(* CODESYS project SPT_NC_Homing.library
   Company: Beckhoff Automation LLC
   DefaultNamespace: SPT_NCHoming
   Version: 3.0.1
   Placeholder: SPT NC Homing
   Title: SPT NC Homing

Project tree, tasks and I/O mapping:
  libraries: SPT Base Types, * (Beckhoff Automation LLC); SPT NC Axis, * (Beckhoff Automation LLC); Tc2_MC2, * (Beckhoff Automation GmbH); Tc2_Standard, * (Beckhoff Automation GmbH); Tc3_MC2_AdvancedHoming, * (Beckhoff Automation GmbH); Tc3_Module, * (Beckhoff Automation GmbH); Tc3_System, * (Beckhoff Automation GmbH)
  DUTs/
    data type ST_AbsHomeParameters
    data type ST_StepBlockLagBasedParameters
  Function Blocks/
    function block FB_HomeRoutine_AbsHoming [ST]: Axis, CyclicLogic, Execute, Parameters
    function block FB_HomeRoutine_HardStop [ST]: Axis, CyclicLogic, Execute, HomePosition, Parameters
    function block FB_HomeRoutine_SetPosition [ST]: Axis, CyclicLogic, Execute, HomePosition
    function block FB_HomeRoutine_SetZeroHere [ST]: Axis, CyclicLogic, Execute
  Project Information/
    function F_GetCompany [ST]
    function F_GetTitle [ST]
    function F_GetVersion [ST]
  Version/
    global variables Global_Version
*)

// DUTs/ST_AbsHomeParameters
TYPE ST_AbsHomeParameters :
    STRUCT
        PositionBias           : LREAL;
        PositionLimit_Positive : LREAL;
        PositionLimit_Negative : LREAL;
    END_STRUCT
END_TYPE

// DUTs/ST_StepBlockLagBasedParameters
TYPE ST_StepBlockLagBasedParameters :
    STRUCT
        Direction              : MC_Home_Direction := mcNegativeDirection;
        Velocity               : LREAL             := 10;
        Acceleration           : LREAL             := 100;
        Deceleration           : LREAL             := 100;
        Jerk                   : LREAL             := 1000;
        DetectionVelocityLimit : LREAL             := 5;
        DetectionVelocityTime  : TIME              := T#500MS;
        TimeLimit              : TIME;
        DistanceLimit          : LREAL;
        TorqueLimit            : LREAL            := 10;
        LagLimit               : LREAL            := 10;
        Options                : ST_Home_Options3 := (InstantLagReduction := TRUE);
    END_STRUCT
END_TYPE

// Version/Global_Version
{attribute 'TcGenerated'}
{attribute 'no-analysis'}
{attribute 'linkalways'}
// This function has been automatically generated from the project information.
VAR_GLOBAL CONSTANT
	{attribute 'const_non_replaced'}
	stLibVersion_SPT_NC_Homing : ST_LibVersion := (iMajor := 3, iMinor := 0, iBuild := 1, iRevision := 0, nFlags := 1, sVersion := '3.0.1');
END_VAR

// Function Blocks/FB_HomeRoutine_AbsHoming
FUNCTION_BLOCK FB_HomeRoutine_AbsHoming EXTENDS FB_CyclicFB IMPLEMENTS I_MotionSequence
VAR
    _Axis : I_BasicAxis;
END_VAR

VAR
    _HomingDn                 : BOOL;
    _Reset                    : BOOL;
    _Parameters               : REFERENCE TO ST_AbsHomeParameters;
    SequenceStep              : UDINT;
    ReadWatchdog              : TON;
    WriteWatchdog             : TON;
    McReadParameter_Bias      : MC_ReadParameter;
    McWriteParameter_Bias     : MC_WriteParameter;
    McWriteParameter_SwPosLim : MC_WriteParameter;
    McWriteParameter_SwNegLim : MC_WriteParameter;
    McHome                    : MC_Home;
    CurrentPositionBias       : LREAL;
END_VAR

//There should be no code in the function block body

PROPERTY Axis : I_BasicAxis
GET
Axis := _Axis;
END_GET
SET
_Axis := Axis;
END_SET
END_PROPERTY

METHOD CyclicLogic
VAR_INPUT
END_VAR
IF __ISVALIDREF(_Parameters) THEN
    CASE SequenceStep OF
        0: (* Init State *)
            _Busy                             := TRUE;
            ReadWatchdog.IN                   := FALSE;
            WriteWatchdog.IN                  := TRUE;
            McReadParameter_Bias.Enable       := FALSE;
            McWriteParameter_Bias.Execute     := TRUE;
            McWriteParameter_SwPosLim.Execute := TRUE;
            McWriteParameter_SwNegLim.Execute := TRUE;
            SequenceStep                      := 10;
        10: (* Wait for init done *)

            // check for errors
            IF WriteWatchdog.Q THEN
                SequenceStep := 500;
                _Error       := TRUE;
                _ErrorID     := 10;
            ELSIF McWriteParameter_Bias.Error THEN
                SequenceStep := 500;
                _Error       := TRUE;
                _ErrorID     := McWriteParameter_Bias.ErrorID;
            ELSIF McWriteParameter_SwPosLim.Error THEN
                SequenceStep := 500;
                _Error       := TRUE;
                _ErrorID     := McWriteParameter_SwPosLim.ErrorID;
            ELSIF McWriteParameter_SwNegLim.Error THEN
                SequenceStep := 500;
                _Error       := TRUE;
                _ErrorID     := McWriteParameter_SwNegLim.ErrorID;
            END_IF

            IF (McWriteParameter_Bias.Done AND McWriteParameter_SwPosLim.Done AND McWriteParameter_SwNegLim.Done) THEN
                WriteWatchdog.IN := FALSE;
                McHome.Execute   := TRUE;
                _Busy            := FALSE;
            END_IF
        20: (* Reads the Position Bias Variable *)
            _Busy                             := TRUE;
            WriteWatchdog.IN                  := FALSE;
            McWriteParameter_Bias.Execute     := FALSE;
            McWriteParameter_SwPosLim.Execute := FALSE;
            McWriteParameter_SwNegLim.Execute := FALSE;

            (* 1042 = Axis Encoder Offset ... AKA: Position Bias *)
            IF NOT McReadParameter_Bias.Enable THEN
                ReadWatchdog.IN             := TRUE;
                McReadParameter_Bias.Enable := TRUE;
            END_IF

            IF (McReadParameter_Bias.Enable AND McReadParameter_Bias.Valid) THEN
                ReadWatchdog.IN             := FALSE;
                McReadParameter_Bias.Enable := FALSE;

                (* Do the calculations to figure how far to adjust the Position Bias # *)

                (* Write Value back to the bias for the new teach position *)
                _Parameters.PositionBias := CurrentPositionBias + (_Axis.Axis.NcToPlc.ActPos * -1.0);
                SequenceStep             := 30;
            ELSIF McReadParameter_Bias.Error THEN
                SequenceStep := 500;
                _Error       := TRUE;
                _ErrorID     := McReadParameter_Bias.ErrorID;
            ELSIF ReadWatchdog.Q THEN
                SequenceStep := 500;
                _Error       := TRUE;
                _ErrorID     := 20;
            END_IF
        30:
            _Busy                             := TRUE;
            WriteWatchdog.IN                  := TRUE;
            McWriteParameter_Bias.Execute     := TRUE;
            McWriteParameter_SwPosLim.Execute := TRUE;
            McWriteParameter_SwNegLim.Execute := TRUE;
            SequenceStep                      := 10;
        500: (* Error State *)
            _Busy                             := FALSE;
            ReadWatchdog.IN                   := FALSE;
            WriteWatchdog.IN                  := FALSE;
            McReadParameter_Bias.Enable       := FALSE;
            McWriteParameter_Bias.Execute     := FALSE;
            McWriteParameter_SwPosLim.Execute := FALSE;
            McWriteParameter_SwNegLim.Execute := FALSE;
    END_CASE
ELSE
    _Busy                             := FALSE;
    _Error                            := FALSE;
    _ErrorID                          := 0;
    SequenceStep                      := 0;
    ReadWatchdog.IN                   := FALSE;
    WriteWatchdog.IN                  := FALSE;
    McReadParameter_Bias.Enable       := FALSE;
    McWriteParameter_Bias.Execute     := FALSE;
    McWriteParameter_SwPosLim.Execute := FALSE;
    McWriteParameter_SwNegLim.Execute := FALSE;
END_IF

ReadWatchdog(PT := T#1S);
WriteWatchdog(PT := T#1S);
McHome(Axis := _Axis.Axis, HomingMode := MC_ForceCalibration);

(* Position Bias Reading *)
McReadParameter_Bias(ParameterNumber := MC_AxisParameter.AxisEncoderOffset, (*AxisEncoderOffset*)
                     Axis            := _Axis.Axis,
                     Value           => CurrentPositionBias);

(* Writes the Position Bias Variable *)
McWriteParameter_Bias(Execute         := McWriteParameter_Bias.Execute,
                      ParameterNumber := MC_AxisParameter.AxisEncoderOffset, (*AxisEncoderOffset*)
                      Value           := _Parameters.PositionBias,
                      Axis            := _Axis.Axis);

(* Writes the SW Positive Limit Variable *)
McWriteParameter_SwPosLim(Execute         := McWriteParameter_SwPosLim.Execute,
                          ParameterNumber := MC_AxisParameter.SWLimitPos,
                          Value           := _Parameters.PositionLimit_Positive,
                          Axis            := _Axis.Axis);

(* Writes the SW Negetive Limit Variable *)
McWriteParameter_SwNegLim(Execute         := McWriteParameter_SwNegLim.Execute,
                          ParameterNumber := MC_AxisParameter.SWLimitNeg,
                          Value           := _Parameters.PositionLimit_Negative,
                          Axis            := _Axis.Axis);
END_METHOD

METHOD Execute : BOOL
IF (_Axis = 0) OR _Busy OR NOT (McWriteParameter_Bias.Done AND McWriteParameter_SwPosLim.Done AND McWriteParameter_SwNegLim.Done) THEN
    RETURN;
END_IF

_Busy        := TRUE;
_Error       := FALSE;
_ErrorID     := 0;
_HomingDn    := FALSE;
SequenceStep := 20;
Execute      := TRUE;
END_METHOD

PROPERTY Parameters : REFERENCE TO ST_AbsHomeParameters
GET
IF __ISVALIDREF(_Parameters) THEN
    Parameters REF= _Parameters;
END_IF
END_GET
SET
_Parameters ref= Parameters;
END_SET
END_PROPERTY

END_FUNCTION_BLOCK

// Function Blocks/FB_HomeRoutine_HardStop
FUNCTION_BLOCK FINAL FB_HomeRoutine_HardStop EXTENDS FB_CyclicFB IMPLEMENTS I_MotionSequence
VAR
    _Axis : I_BasicAxis;
END_VAR

VAR
    MCStepBlock    : MC_StepBlockLagBasedDetection;
    MCHomeDirect   : MC_HomeDirect;
    MCReset        : MC_Reset;
    MCAbortHoming  : MC_AbortHoming;
    AxisParameters : MC_HomingParameter;
    _Parameters    : ST_StepBlockLagBasedParameters;
    _HomePosition  : LREAL;
    SequenceStep   : UDINT;
END_VAR

//There should be no code in the function block body

PROPERTY Axis : I_BasicAxis
GET
Axis := _Axis;
END_GET
SET
_Axis := Axis;
END_SET
END_PROPERTY

METHOD PUBLIC CyclicLogic
CASE SequenceStep OF
    10:
        MCStepBlock(Axis                   := _Axis.Axis,
                    Parameter              := AxisParameters,
                    Execute                := TRUE,
                    Direction              := _Parameters.Direction,
                    Velocity               := _Parameters.Velocity,
                    Acceleration           := _Parameters.Acceleration,
                    Deceleration           := _Parameters.Deceleration,
                    Jerk                   := _Parameters.Jerk,
                    DetectionVelocityLimit := _Parameters.DetectionVelocityLimit,
                    DetectionVelocityTime  := _Parameters.DetectionVelocityTime,
                    TimeLimit              := _Parameters.TimeLimit,
                    DistanceLimit          := _Parameters.DistanceLimit,
                    TorqueLimit            := _Parameters.TorqueLimit,
                    LagLimit               := _Parameters.LagLimit,
                    Options                := _Parameters.Options);

        IF NOT MCStepBlock.Busy THEN
            IF MCStepBlock.Error THEN
                _Error       := TRUE;
                _ErrorID     := MCStepBlock.ErrorID;
                SequenceStep := 999;
            ELSE
                //No error occurred
                SequenceStep := SequenceStep + 10;
            END_IF

            MCStepBlock(Axis := _Axis.Axis, Parameter := AxisParameters, Execute := FALSE);
        END_IF
    20:
        MCHomeDirect(Axis        := _Axis.Axis,
                     Parameter   := AxisParameters,
                     Execute     := TRUE,
                     SetPosition := _HomePosition);

        IF NOT MCHomeDirect.Busy THEN
            IF MCHomeDirect.Error THEN
                _Error       := TRUE;
                _ErrorID     := MCHomeDirect.ErrorID;
                SequenceStep := 999;
            END_IF

            //Done
            SequenceStep := 0;
            MCHomeDirect(Axis := _Axis.Axis, Parameter := AxisParameters, Execute := FALSE);
        END_IF
    999:
        //An error occurred above--clear out position lag so we don't fault the axis with AbortHoming
        MCReset(Axis := _Axis.Axis, Execute := TRUE);
        IF NOT MCReset.Busy THEN
            //If this errors there's not much we can do about it
            SequenceStep := 1000;
            MCReset(Axis := _Axis.Axis, Execute := FALSE);
        END_IF
    1000:
        MCAbortHoming(Axis := _Axis.Axis, Parameter := AxisParameters, Execute := TRUE);
        IF NOT MCAbortHoming.Busy THEN
            IF MCAbortHoming.Error THEN
                _Error       := TRUE;
                _ErrorID     := MCAbortHoming.ErrorID;
                SequenceStep := 0;
            ELSE
                //No error occurred
                SequenceStep := 0;
            END_IF

            MCAbortHoming(Axis := _Axis.Axis, Parameter := AxisParameters, Execute := FALSE);
        END_IF
END_CASE

_Busy := SequenceStep <> 0;
END_METHOD

METHOD PUBLIC Execute : BOOL
IF (_Axis = 0) OR _Busy THEN
    RETURN;
END_IF

_Busy        := TRUE;
_Error       := FALSE;
_ErrorID     := 0;
SequenceStep := 10;
Execute      := TRUE;
END_METHOD

PROPERTY HomePosition : LREAL
GET
HomePosition := _HomePosition;
END_GET
SET
_HomePosition := HomePosition;
END_SET
END_PROPERTY

PROPERTY Parameters : ST_StepBlockLagBasedParameters
GET
Parameters := _Parameters;
END_GET
SET
_Parameters := Parameters;
END_SET
END_PROPERTY

END_FUNCTION_BLOCK

// Function Blocks/FB_HomeRoutine_SetPosition
FUNCTION_BLOCK FINAL FB_HomeRoutine_SetPosition EXTENDS FB_CyclicFB IMPLEMENTS I_MotionSequence
VAR_INPUT
END_VAR

VAR_OUTPUT
END_VAR

VAR
    _Axis : I_BasicAxis;
END_VAR

VAR
    MCSetPosition : MC_SetPosition;
END_VAR

//There should be no code in the function block body

PROPERTY Axis : I_BasicAxis
GET
Axis := _Axis;
END_GET
SET
_Axis := Axis;
END_SET
END_PROPERTY

METHOD PUBLIC CyclicLogic
MCSetPosition(Axis := _Axis.Axis, Busy => _Busy);
IF NOT MCSetPosition.Busy THEN
    IF MCSetPosition.Error THEN
        _Error   := TRUE;
        _ErrorID := MCSetPosition.ErrorID;
    END_IF

    MCSetPosition(Axis := _Axis.Axis, Execute := FALSE);
END_IF
END_METHOD

METHOD PUBLIC Execute : BOOL
IF (_Axis = 0) THEN
    RETURN;
END_IF

MCSetPosition(Axis := _Axis.Axis, Execute := TRUE, Mode := FALSE);
_Error   := FALSE;
_ErrorID := 0;
Execute  := TRUE;
END_METHOD

PROPERTY HomePosition : LREAL
GET
HomePosition := MCSetPosition.Position;
END_GET
SET
MCSetPosition.Position := HomePosition;
END_SET
END_PROPERTY

END_FUNCTION_BLOCK

// Function Blocks/FB_HomeRoutine_SetZeroHere
FUNCTION_BLOCK FINAL FB_HomeRoutine_SetZeroHere EXTENDS FB_CyclicFB IMPLEMENTS I_MotionSequence
VAR_INPUT
END_VAR

VAR_OUTPUT
END_VAR

VAR
    _Axis : I_BasicAxis;
END_VAR

VAR
    MCSetPosition : MC_SetPosition;
END_VAR

//There should be no code in the function block body

PROPERTY Axis : I_BasicAxis
GET
Axis := _Axis;
END_GET
SET
_Axis := Axis;
END_SET
END_PROPERTY

METHOD PUBLIC CyclicLogic
MCSetPosition(Axis := _Axis.Axis, Busy => _Busy);
IF NOT MCSetPosition.Busy THEN
    IF MCSetPosition.Error THEN
        _Error   := TRUE;
        _ErrorID := MCSetPosition.ErrorID;
    END_IF

    MCSetPosition(Axis := _Axis.Axis, Execute := FALSE);
END_IF
END_METHOD

METHOD PUBLIC Execute : BOOL
IF (_Axis = 0) THEN
    RETURN;
END_IF

MCSetPosition(Axis     := _Axis.Axis,
              Execute  := TRUE,
              Position := 0.0,
              Mode     := FALSE);

_Error   := FALSE;
_ErrorID := 0;
Execute  := TRUE;
END_METHOD

END_FUNCTION_BLOCK

// Project Information/F_GetCompany
// This function has been automatically generated from the project information.
{attribute 'signature_flag' := '1073741824'}
{attribute 'TcGenerated'}
{attribute 'no-analysis'}
FUNCTION F_GetCompany : WSTRING
VAR_INPUT
	
END_VAR

F_GetCompany := "Beckhoff Automation LLC";

END_FUNCTION

// Project Information/F_GetTitle
// This function has been automatically generated from the project information.
{attribute 'signature_flag' := '1073741824'}
{attribute 'TcGenerated'}
{attribute 'no-analysis'}
FUNCTION F_GetTitle : WSTRING
VAR_INPUT
	
END_VAR

F_GetTitle := "SPT NC Homing";

END_FUNCTION

// Project Information/F_GetVersion
// This function has been automatically generated from the project information.
{attribute 'signature_flag' := '1073741824'}
{attribute 'TcGenerated'}
{attribute 'no-analysis'}
FUNCTION F_GetVersion : ST_LibVersion
VAR_INPUT
	
END_VAR

F_GetVersion.iMajor := 3;
F_GetVersion.iMinor := 0;
F_GetVersion.iBuild := 1;
F_GetVersion.iRevision := 0;
F_GetVersion.sVersion := '3.0.1';
F_GetVersion.nFlags := 1;

END_FUNCTION
